{attribute 'GeneratedUsingTerminal: ELX3181-0000-0016'}
{attribute addProperty BoxType "ELX3181-0000-0016"}
{attribute addProperty Id "EtcSlaveTerminalBaseCh_1Ch_1_A1FAE75910WcStateAT %I*WcState_9091E0EB2InfoDataAT %I*InfoData_90184F0C16"}
{attribute addProperty CRC "1508372664"}
{attribute addProperty Size "28"}
TYPE ELX3181_59E7F0B8 EXTENDS EtcSlaveTerminalBase :
STRUCT
	{attribute addProperty Name "Ch_1"}
	Ch_1 : Ch_1_A1FAE759;
	{attribute addProperty Name "WcState"}
	WcState : WcState_9091E0EB;
	{attribute addProperty Name "InfoData"}
	InfoData : InfoData_90184F0C;
END_STRUCT
END_TYPE

(* stored: Version 1.2.0.0, ProductVersion 3.1.4024.9
   DUT ELX3181_59E7F0B8: Id {dbcff17a-4ca7-4cc4-8d22-bbe8a2ab8a62} *)
